// TIA Portal V17 export
// export: Created 2024-08-09T12:53:17.3488497Z, ExportSetting WithDefaults, DisplayName Totally Integrated Automation Portal, DisplayVersion V17 Update 7, DisplayName TIA Portal Openness, DisplayVersion V17 Update 7, DisplayName TIA Portal Version Control Interface, DisplayVersion V17, DisplayName STEP 7 Professional, DisplayVersion V17 Update 7, DisplayName STEP 7 Safety, DisplayVersion V17 Update 6, DisplayName WinCC Professional, DisplayVersion V17 Update 7
TYPE "S_Lots_Tache"
// stored: IsFailsafeCompliant false
   STRUCT
      Zones_Suiv { ExternalAccessible := 'False'; ExternalVisible := 'False'; ExternalWritable := 'False'} : Array[0.."Nbr_Max_Lots"] of SInt;
   END_STRUCT;
   // Zones_Suiv[0..19] := -1;
END_TYPE
